INTERFACE I_AlarmObserver

METHOD PUBLIC cleared : BOOL		// Called when an alarm is cleared
VAR_INPUT
	iAlarm:	ST_CLEAR_ALARM;
END_VAR
END_METHOD

METHOD PUBLIC raised : BOOL		// Called when an alarm is raised
VAR_INPUT
	iAlarm:	ST_ACTIVE_ALARM;
END_VAR
END_METHOD

END_INTERFACE

(* stored: Version 1.1.0.1, ProductVersion 3.1.4026.18
   Itf I_AlarmObserver: Id {6214b008-3d2a-4036-9865-3bdc776e05d3}
   Method cleared: Id {049a4742-3584-4315-b7f4-ca80395e483b}
   Method raised: Id {b89b7ab5-32d1-4c11-a722-7141613373a0} *)
